FUNCTION_BLOCK FB_TopElement1_HMI EXTENDS FB_BaseTopElement_HMI IMPLEMENTS ITF_TopElement1_HMI
VAR
	itfTopElementConnector			: ITF_TopElement1_HMI_Connector;
	refstTopElementData				: REFERENCE TO ST_TopElement1_HMI;
	
	itfGE1							: ITF_GroupE_TE1_HMI;
	
	itfCE1							: ITF_ControlE_TE1_HMI;
	itfCE2							: ITF_ControlE_TE1_HMI;
	
	itfC1							: ITF_Component_TE1_HMI;
	itfC2							: ITF_Component_TE1_HMI;
	itfC3							: ITF_Component_TE1_HMI;
END_VAR

METHOD FB_init : BOOL
VAR_INPUT
	bInitRetains : BOOL; // if TRUE, the retain variables are initialized (warm start / cold start)
	bInCopyCode : BOOL;  // if TRUE, the instance afterwards gets moved into the copy code (online change)
	itfBaseLoggerConnector				: ITF_BaseLogger_HMI_Connector;	//bezpośredni łącznik do logera
	itfTopElementConnector				: ITF_TopElement1_HMI_Init;
	itfGE1								: ITF_GroupE_TE1_HMI;
	itfCE1								: ITF_ControlE_TE1_HMI;
	itfCE2								: ITF_ControlE_TE1_HMI;
	itfC1								: ITF_Component_TE1_HMI;
	itfC2								: ITF_Component_TE1_HMI;
	itfC3								: ITF_Component_TE1_HMI;
END_VAR
//Przypisanie do elementu który własnie stworzyliśmy
THIS^.itfTopElementConnector			:= itfTopElementConnector;
//Przypisanie do elementów z biblioteki
THIS^.itfBaseLoggerElementConnector		:= itfTopElementConnector;
THIS^.itfBaseComponentConnector			:= itfTopElementConnector;
THIS^.itfBaseControlElementConnector	:= itfTopElementConnector;
THIS^.itfBaseGroupElementConnector		:= itfTopElementConnector;
THIS^.itfBaseTopElementConnector		:= itfTopElementConnector;
//
THIS^.itfBaseLoggerConnector			:= itfBaseLoggerConnector;

THIS^.AddControlElement (itfControlElementHMI := itfGE1);
THIS^.itfGE1 := itfGE1;

THIS^.AddControlElement (itfControlElementHMI := itfCE1);
THIS^.itfCE1 := itfCE1;

THIS^.AddControlElement (itfControlElementHMI := itfCE2);
THIS^.itfCE2 := itfCE2;

THIS^.AddComponent (itfComponentHMI := itfC1);
THIS^.itfC1 := itfC1;

THIS^.AddComponent (itfComponentHMI := itfC2);
THIS^.itfC2 := itfC2;

THIS^.AddComponent (itfComponentHMI := itfC3);
THIS^.itfC3 := itfC3;

IF (THIS^.itfTopElementConnector <> 0 AND
	THIS^.itfBaseLoggerElementConnector <> 0 AND
	THIS^.itfBaseComponentConnector	<> 0 AND
	THIS^.itfBaseControlElementConnector <> 0 AND
	THIS^.itfBaseGroupElementConnector <> 0 AND
	THIS^.itfBaseTopElementConnector <> 0 AND
	THIS^.itfBaseLoggerConnector <> 0) THEN
	THIS^.bIsInit						:= TRUE;
END_IF
END_METHOD

METHOD LinkTopElementData : BOOL
VAR_INPUT
	stData				: REFERENCE TO ST_TopElement1_HMI_Link;
END_VAR

VAR
	stBaseGroupElem: INT;
END_VAR
THIS^.refstTopElementData REF= stData.stTopElement;

THIS^.refstBaseLoggerElementDataHMI REF= stData.stBaseLoggerElement;
THIS^.refstBaseComponentDataHMI REF= stData.stBaseComponent;
THIS^.refstBaseControlElementDataHMI REF= stData.stBaseControlElement;
THIS^.refstBaseGroupElementDataHMI REF= stData.stBaseGroupElement;
THIS^.refstBaseTopElementDataHMI REF= stData.stBaseTopElement;

THIS^.itfGE1.LinkGroupEData (stData := stData.stGE1);

THIS^.itfCE1.LinkControlEData (stData := stData.stCE1);
THIS^.itfCE2.LinkControlEData (stData := stData.stCE2);

THIS^.itfC1.LinkComponentData (stData := stData.stC1);
THIS^.itfC2.LinkComponentData (stData := stData.stC2);
THIS^.itfC3.LinkComponentData (stData := stData.stC3);

(*
THIS^.itfControlElement1.LinkControlElementData (stData := stData.stControlElement1);
THIS^.itfControlElement2.LinkControlElementData (stData := stData.stControlElement2);
THIS^.itfGroupElement1.LinkGroupelementData (stData := stData.stGroupElement1);
THIS^.itfComponent1.LinkComponentData (stData := stData.stComponent1);
THIS^.itfComponent2.LinkComponentData (stData := stData.stComponent2);
THIS^.itfComponent3.LinkComponentData (stData := stData.stComponent3);
*)
THIS^.CreateLinkToEventsMemory ();

IF (__ISVALIDREF (THIS^.refstTopElementData) AND this^.IsLinkedReferences ()) THEN
	THIS^.bIsValidData		:= TRUE;
	LinkTopElementData		:= TRUE;
END_IF
END_METHOD

END_FUNCTION_BLOCK

(* stored: Version 1.1.0.1, ProductVersion 3.1.4024.15
   POU FB_TopElement1_HMI: Id {72240472-9116-03cb-36c6-17374bd97d62}, SpecialFunc None
   Folder ITF_NazwaPB_HMI: Id {ff441856-cda9-0c25-0700-4cb0f490f4a3}
   Method FB_init: Id {1625a283-a5a4-0658-16db-29129ffd0296}
   Method LinkTopElementData: Id {b5b619bd-8b68-4908-b96b-4f1ab05bb941} *)
